(*~
	<docu>
		<summary>
			Completes the execution of the current step and moves the sequencer pointer to the next step in order of execution.
			The call returns ```ITcoObjectRestorer``` that allows to restore object upon step completition.
		</summary>		
		<returns></returns>	
	</docu>	
~*)
METHOD PROTECTED FINAL CompleteStep : ITcoObjectRestorer
_theOrderOfTheCurrentlyExecutedStep := _theOrderOfTheCurrentlyExecutedStep + 1;	
_currentStep.Status := eStepStatus.Done;
OnStepCompleted();
_modeController._stepIn.DoneWhen(_modeController._stepIn.Execute());
CompleteStep := THIS^;
END_METHOD

(*~
	<docu>
		<summary>
			Gets the information about the current step.						
		</summary>				
	</docu>	
~*)
PROPERTY CurrentStep : REFERENCE TO StepDetails
GET
CurrentStep REF= _currentStep;
END_GET
END_PROPERTY

METHOD FB_init : BOOL
VAR_INPUT
	bInitRetains : BOOL; // if TRUE, the retain variables are initialized (warm start / cold start)
	bInCopyCode : BOOL;  // if TRUE, the instance afterwards gets moved into the copy code (online change)
	Parent : ITcoObject;
	AutoRestoreMode : eRestoreMode; 
END_VAR
SUPER^.FB_init(bInitRetains, bInCopyCode, Parent, AutoRestoreMode);
END_METHOD

(*~
	<docu>
		<summary>
			Performs the check of the uniqueness of ```inStepId``` in the sequence.
			<remarks>			
				<note type="important">
					The StepId of each step in the sequence must be unique throughout the complete sequence, and it must not be changed.
				</note>
			</remarks>			
		</summary>				
	</docu>	
~*)
METHOD PRIVATE IsStepIdUnique
VAR_INPUT
(*~
	<docu>
		<summary>
			StepId to be checked for uniqueness.
		</summary>				
	</docu>	
~*)
	inStepID : INT;
END_VAR
VAR
	_i	: UINT;
	_hiIndex : UINT;
	_pUid : INT;
    _pNewSteps : POINTER TO INT;		
	_message : STRING(254);
END_VAR
IF ((_numberOfStepsInSequence <> _previousNumberOfStepsInSequence) AND _previousNumberOfStepsInSequence > 0) AND _stepIdUniquenessChecked AND NOT _sequencerHasError THEN
	_stepIdUniquenessChecked := FALSE;
	_previousNumberOfStepsInSequence := 0;
	_stepCounter := 0;
	_numberOfStepsInSequence := 0;
END_IF

IF NOT _stepIdUniquenessChecked AND NOT _sequencerHasError THEN

	// Increment order of the currently controlled step
	_theOrderOfTheCurrentlyEvaluatedStep := _theOrderOfTheCurrentlyEvaluatedStep + 1;
	
	IF(_stepCounter < _theOrderOfTheCurrentlyEvaluatedStep) THEN
		_stepCounter := _theOrderOfTheCurrentlyEvaluatedStep;
		_stepCounter := _stepCounter - 1; 
	END_IF
	
	_numberOfStepsInSequence := _stepCounter;
	
	IF (_numberOfStepsInSequence = _previousNumberOfStepsInSequence) AND (_numberOfStepsInSequence > 0) AND NOT _stepIdUniquenessChecked AND NOT _sequencerHasError THEN
		IF (_pPreviusSteps <> 0) THEN
			__DELETE(_pPreviusSteps);
		END_IF
		IF (_pNewSteps <> 0) THEN
			__DELETE(_pNewSteps);
		END_IF	
		_stepIdUniquenessChecked := TRUE;
		_theOrderOfTheCurrentlyEvaluatedStep := 0;
		_theOrderOfTheCurrentlyExecutedStep := 0;
		RETURN;		
	END_IF
	
	//Stores first StepId		
	IF (_numberOfStepsInSequence = 0) THEN
		//It should not exists, if yes delete and create again
		IF (_pPreviusSteps <> 0) THEN
			__DELETE(_pPreviusSteps);
		END_IF
		_pPreviusSteps := __NEW(UINT, 1);
		_pPreviusSteps[0] := inStepID;
	ELSE
		IF (_pNewSteps <> 0) THEN
			__DELETE(_pNewSteps);
		END_IF
		_pNewSteps := __NEW(UINT, (_numberOfStepsInSequence+1));

		//Compare with previous Steps and copy previous Steps to new array
		_hiIndex := _numberOfStepsInSequence-1;
		FOR _i := 0 TO _hiIndex DO
			_pUid := _pPreviusSteps[_i];
			IF inStepID = _pUid THEN
				IF NOT _sequencerHasError THEN
					IF (_pPreviusSteps <> 0) THEN
						__DELETE(_pPreviusSteps);
					END_IF	
					IF (_pNewSteps <> 0) THEN
						__DELETE(_pNewSteps);
					END_IF
					_sequencerErrorId := eSequencerError.NotUniqueStepId;
					_message := CONCAT('ERROR NOT UNIQUE STEP_ID ',UINT_TO_STRING(inStepID));
					_currentStep.Description := _message;
					_currentStep.Status := eStepStatus.Error;
					THIS^.Messenger.Post(_message, eMessageCategory.ProgrammingError);
					_sequencerHasError := TRUE;
					RETURN;					
				END_IF
			ELSE
				_pNewSteps[_i] := _pPreviusSteps[_i];
			END_IF
		END_FOR
		//Store new StepId
		_pNewSteps[_numberOfStepsInSequence] := inStepID;
		//Delete and create again
		IF (_pPreviusSteps <> 0) THEN
			__DELETE(_pPreviusSteps);
		END_IF		
		_pPreviusSteps :=  __NEW(UINT, (_numberOfStepsInSequence+1));
		//Copy
		_hiIndex := _hiIndex+1;
		FOR _i := 0 TO _hiIndex DO
			_pPreviusSteps[_i] := _pNewSteps[_i];			
		END_FOR

		IF (_pNewSteps <> 0) THEN
			__DELETE(_pNewSteps);
		END_IF
	END_IF	
END_IF
IF _stepIdUniquenessChecked THEN
	IF (_pPreviusSteps <> 0) THEN
		__DELETE(_pPreviusSteps);
	END_IF
	IF (_pNewSteps <> 0) THEN
		__DELETE(_pNewSteps);
	END_IF
END_IF
END_METHOD

(*~
	<docu>
		<summary>
			Main method of the sequener. Custom code needs to be placed here. The sequencer is executed by call of InstanceName.Run() method.
			This method is abstract, and it must be overridden in derived block.
		</summary>
	</docu>
~*)
METHOD PROTECTED ABSTRACT Main : BOOL
END_METHOD

(*~
	<docu>
		<summary>
			Handles changing the sequencer mode (Cyclic, Step).
		</summary>
	</docu>
~*)
PROPERTY ModeController : ITcoSequencerModeController
GET
ModeController := _modeController;
END_GET
END_PROPERTY

(*~
	<docu>
		<summary>
			Ensures that after each download, StepId uniqueness check is performed. 
			<remarks>			
				<note type="important">
					Do not call this method explicitly.
				</note>
			</remarks>		
		</summary>			
	</docu>	
~*)
{attribute 'call_after_online_change_slot' := '200'}
METHOD PRIVATE OnlineChange
_stepIdUniquenessChecked := FALSE;

_stepCounter := 0;
_numberOfStepsInSequence := 0;
_previousNumberOfStepsInSequence := 0;
END_METHOD


(*~
	<docu>
		<summary>
			This method is called on sequence completion (the sequencer's last step was completed). 
			This method can be overridden in derived block with a custom logic.
		</summary>			
	</docu>	
~*)
METHOD PROTECTED OnSequenceCompleted
END_METHOD

(*~
	<docu>
		<summary>
			This method is called when sequence enters error state. The method is called until the error is cleared. 
			This method can be overridden in derived block with a custom logic.
		</summary>			
	</docu>	
~*)
METHOD PROTECTED OnSequencerError
VAR_INPUT
	inErrorId : eSequencerError;
END_VAR
END_METHOD

(*~
	<docu>
		<summary>
			This method is executed upon step completion.
			This method can be overridden in derived block by custom logic.
		</summary>			
	</docu>	
~*)
METHOD PROTECTED OnStepCompleted
END_METHOD

(*~
	<docu>
		<summary>
			Implicit calling of this method is ensured by calling the method Run().
			It must not be called explicitely by consumer code in derived blocks.
			<remarks>			
				<note type="important">
					Do not call this method explicitly.
				</note>
			</remarks>
		</summary>			
	</docu>	
~*)
METHOD INTERNAL FINAL Open
VAR
	_message	:	STRING(254);
END_VAR
_theOrderOfTheCurrentlyEvaluatedStep := 0;

IF _requestStepActive AND _requestedStepId <> MinStepID AND (_modeController.Mode <> eSequencerMode.StepMode OR _modeController._stepIn.Busy OR _checkStepIdRequestedInStepMode) THEN
	_requestStepCycle := _requestStepCycle +1;
ELSE
	_requestStepCycle := 0;
END_IF

IF _requestStepCycle > 1 AND NOT _sequencerHasError THEN
	_sequencerErrorId := eSequencerError.StepWithRequestedIdDoesNotExists;
	_message := CONCAT('REQUESTED STEP_ID: ',UINT_TO_STRING(_requestedStepId));
	_message := CONCAT(_message, ' DOES NOT EXIST');
	_currentStep.Description := _message;
	_currentStep.Status := eStepStatus.Error;
	THIS^.Messenger.Post(_message, eMessageCategory.ProgrammingError);
	_sequencerHasError := TRUE;
END_IF

//???? Check if needs to be here.
IF _sequencerHasError AND (_sequencerErrorId = eSequencerError.NotUniqueStepId) THEN
	_sequencerErrorId := eSequencerError.noerror;	
	_sequencerHasError := FALSE;
	_stepIdUniquenessChecked := FALSE;
	_numberOfStepsInSequence := 0;
	_stepCounter := 0;
	_previousNumberOfStepsInSequence := 0;
END_IF

_restoringSequence := FALSE;
END_METHOD

(*~
	<docu>
		<summary>
			Terminates the currently executed step and set the sequencer's pointer to the step with Id that corresponds to ```inRequestedStepID``` parameter.
			When the order of the requested step is higher than the order of the currently finished step (the requested step is "after" the current one)
			the requested step is started in the same context cycle.
			When the order of the requested step is lower than the order of the currently finished step (the requested step is "before" the current one)
			the requested step is started in the next context cycle.
			If the requested step is not found even in the next context cycle, the sequencer enters error state ```StepWithRequestedIdDoesNotExists```.
			<para>
				See <see cref="eSequencerError"/> for detailed description.
			</para>
		</summary>
	</docu>
~*)
METHOD PROTECTED FINAL RequestStep : ITcoSequencer
VAR_INPUT
	(*~
		<docu>
			<summary>
				StepId of the step to be executed.
			</summary>
		</docu>
	~*)
	inRequestedStepID : INT := MinStepID;
END_VAR
VAR
	_message : STRING(254);
END_VAR
_modeController._stepIn.Restore();

_currentStep.Status := eStepStatus.Done;

_checkStepIdRequestedInStepMode := TRUE;

IF(inRequestedStepID <> MinStepID) THEN
	IF _requestedStepId <> MinStepID THEN
		IF NOT  _sequencerHasError THEN
			_sequencerErrorId := eSequencerError.MultipleRequestStepMethodCall;
			_message := CONCAT('REQUESTED STEP_ID: ',UINT_TO_STRING(inRequestedStepID));
			_message := CONCAT(_message, ' HAS BEEN REQUIRED, WHILE PREVIOUS REQUESTED STEP_ID: ');
			_message := CONCAT(_message,UINT_TO_STRING(_requestedStepId));
			_message := CONCAT(_message, ' HAS NOT BEEN YET PERFORMED!');
			_currentStep.Description := _message;
			_currentStep.Status := eStepStatus.Error;
			THIS^.Messenger.Post(_message, eMessageCategory.ProgrammingError);
			_sequencerHasError := TRUE;
		END_IF
	ELSE
		_requestStepCycle := 0;
		_requestedStepId := inRequestedStepID;
		_requestStepActive := TRUE;
	END_IF
END_IF;	

RequestStep := THIS^;
END_METHOD

(*~
	<docu>
		<summary>
			<para>
				This method resets the sequencer. 
				Method is typically called before starting the sequence or after error has occured in the sequence.
			</para>
		</summary>			
	</docu>	
~*)
METHOD PUBLIC Restore : ITcoRestorable
_restoringSequence := TRUE;

StepChanged(0);

_requestStepActive := FALSE;	
_requestedStepId := MinStepID;
_requestStepCycle := 0;
_sequencerHasError := FALSE;
_sequencerErrorId := eSequencerError.noError;
_currentStep.Description := '--------------------------';
_currentStep.ID := 0;
_currentStep.Order := 0;
_currentStep.Status := eStepStatus.None;
_currentStep.Duration := T#0S;

_stepCounter := 0;
_IdOfThePreviouslyExecutedStep := 0;
_numberOfStepsInSequence := 0;
_previousNumberOfStepsInSequence := 0;
_theOrderOfTheCurrentlyExecutedStep := 0;
_theOrderOfThePreviouslyExecutedStep := 0;
_stepIdUniquenessChecked := FALSE;

_StepIdChanged := FALSE;
_StepOrderChanged := FALSE;
_ChangeStepIdFrom := 0;
_ChangeStepIdTo := 0;
_ChangeStepOrderFrom := 0;
_ChangeStepOrderTo := 0;

_StepTimer(IN:= FALSE);

IF _modeController.Mode = eSequencerMode.Invalid THEN
	_modeController.Mode := eSequencerMode.CyclicMode;
END_IF

_modeController._stepForward.Restore();
_modeController._stepBackward.Restore();
_modeController._stepIn.Restore(); 	
_checkStepIdRequestedInStepMode := FALSE;
END_METHOD

(*~
	<docu>
		<summary>
			<para>
				Ensures calling the Open(), Main() and Close() methods in the desired order.
				This method is final, so it cannot be overloaded. The InstanceName.Run() needs to be called cyclically inside the appropriate context.
			</para>
		</summary>			
	</docu>	
~*)
METHOD PUBLIC FINAL Run
THIS^.Open();

_lastActiveCycle := Context.StartCycleCount; 

THIS^.Main();



IF _sequencerHasError THEN
	OnSequencerError(_sequencerErrorId);
END_IF
THIS^.Close();
END_METHOD

(*~
	<docu>
		<summary>
				Step of the sequence. 
		</summary>			
		<returns>
			True when step with given ```StepId``` is in order of the execution; the step is enabled and the sequencer is in the cyclic mode.
			True when step with given ```StepId``` is in order of the execution; the step is enabled, the sequencer is in the step mode and StepIn() method has been triggered.  			
		</returns>			
	</docu>	
~*)
METHOD PROTECTED FINAL Step : BOOL
VAR_INPUT
(*~
	<docu>
		<summary>
			StepId of the current step.
			<remarks>			
				<note type="important">
					This number must be unique throughout the complete sequence.
					It must be a constant or numerical literal and it must not change during the life-time of the sequencer. 
				</note>
			</remarks>
		</summary>		
	</docu>	
~*)
	inStepID				: 	INT;
(*~
	<docu>
		<summary>
			If this value is false, step body is not executed and execution is moved to the next enabled step.
		</summary>				
	</docu>	
~*)
	inEnabled				: 	BOOL;
(*~
	<docu>
		<summary>
			Step description text.
		</summary>				
	</docu>	
~*)
	inStepDescription		: 	STRING(254);		
END_VAR
VAR
	_message 				:	STRING(254);	
	_isInOrderOfExecution 	:	BOOL;	
	_stepModeActive 		: 	BOOL;
	_stepInExecuting 		: 	BOOL;
END_VAR
Step := FALSE;
IF inStepID <= MinStepID THEN
		_message := CONCAT('STEP_ID TOO LOW: ',INT_TO_STRING(inStepID));
		_message := CONCAT(_message, '! MINIMAL VALUE POSSIBLE: ');
		_message := CONCAT(_message,INT_TO_STRING(MinStepID + 1));
		_message := CONCAT(_message,'!!!');
		_currentStep.Description := _message;
		_currentStep.Status := eStepStatus.Error;
		THIS^.Messenger.Post(_message, eMessageCategory.ProgrammingError);
		_sequencerErrorId := eSequencerError.StepIdTooLow;
		_sequencerHasError := TRUE;
ELSIF  inStepID >= MaxStepID THEN
		_message := CONCAT('STEP_ID TOO HIGH: ',INT_TO_STRING(inStepID));
		_message := CONCAT(_message, '! MAXIMAL VALUE POSSIBLE: ');
		_message := CONCAT(_message,INT_TO_STRING(MaxStepID - 1));
		_message := CONCAT(_message,'!!!');
		_currentStep.Description := _message;
		_currentStep.Status := eStepStatus.Error;
		THIS^.Messenger.Post(_message, eMessageCategory.ProgrammingError);
		_sequencerErrorId := eSequencerError.StepIdTooHigh;
		_sequencerHasError := TRUE;
ELSIF NOT _sequencerHasError THEN
	Step := StepInternal(inStepID,inEnabled,inStepDescription);
END_IF;
END_METHOD

(*~
	<docu>
		<summary>
			This method is called at each transition between steps. 
		</summary>			
	</docu>	
~*)
METHOD PRIVATE StepChanged
VAR_INPUT
	newState : INT;
END_VAR
_isFirstStepEntry := TRUE;
_theOrderOfThePreviouslyExecutedStep := 0;
_IdOfThePreviouslyExecutedStep := MinStepID;

_StepTimer(IN:= FALSE);

SUPER^.ChangeStateProtected(newState);
END_METHOD

(*~
	<docu>
		<summary>
			Completes the actually running step, when the ```inCondition``` parameter is ```TRUE```.
			Method is typically called inside a step as the transition method.
		</summary>			
	</docu>	
~*)
METHOD PROTECTED FINAL StepCompleteWhen 
VAR_INPUT
(*~
	<docu>
		<summary>
			The condition under which the step is completed.
		</summary>			
	</docu>	
~*)
	inCondition : BOOL;
END_VAR
IF(inCondition) THEN
	THIS^.CompleteStep();
END_IF
END_METHOD

(*~
	<docu>
		<summary>
				Basic step of the sequence. 
		</summary>			
		<returns>
			True in case when step with given StepId is in order of the execution, the step is enabled and the sequencer is in the cyclic mode.
			True in case when step with given StepId is in order of the execution, the step is enabled, the sequencer is in the step mode and StepIn() method was triggered.  			
		</returns>			
	</docu>	
~*)
METHOD PRIVATE StepInternal : BOOL
VAR_INPUT
(*~
	<docu>
		<summary>
			StepId of the current step.
			<remarks>			
				<note type="important">
					This number must be unique throughout the complete sequence.
					It must be a constant or numerical literal and it must not change during the life-time of the sequencer. 
				</note>
			</remarks>
		</summary>		
	</docu>	
~*)
	inStepID				: 	INT;
(*~
	<docu>
		<summary>
			If this value is false, step body is not executed and execution is moved to the next enabled step.
		</summary>				
	</docu>	
~*)
	inEnabled				: 	BOOL;
(*~
	<docu>
		<summary>
			Step description text.
		</summary>				
	</docu>	
~*)
	inStepDescription		: 	STRING(254);		
END_VAR
VAR
	_message 				:	STRING(254);	
	_isInOrderOfExecution 	:	BOOL;	
	_stepModeActive 		: 	BOOL;
	_stepInExecuting 		: 	BOOL;
END_VAR
IF _modeController.Mode = eSequencerMode.Invalid THEN
	IF NOT _sequencerHasError THEN
		_currentStep.Description := 'INVALID MODE OF THE SEQUENCER!!!';
		_currentStep.Status := eStepStatus.Error;
		THIS^.Messenger.Post('INVALID MODE OF THE SEQUENCER!!!', eMessageCategory.Error);
		_sequencerErrorId := eSequencerError.InvalidSequencerMode;
		_sequencerHasError := TRUE;
	END_IF;		
	RETURN;
END_IF	

//-----------------------------------------------
//     		MULTIPLE CALL REGION
//-----------------------------------------------
// Initialize
StepInternal := FALSE;
_isFirstStepEntry := FALSE;
//-------------------------------------------------------------------------------------------------
//     		Check uniqueness of the StepId
//			If there are even two same StepIds or sequence has not been yet 
//			checked, method return FALSE, so no entrance to the step will be executed
//-------------------------------------------------------------------------------------------------
//-------------------------------------------------------------------------------------------------
//In case of call Restore() in OnStateChange(), this method must exits
//otherwise we get page fault
IF _restoringSequence THEN
	RETURN;
END_IF
IsStepIDUnique(inStepID);
IF NOT _stepIdUniquenessChecked THEN
	_theOrderOfThePreviouslyExecutedStep := -1;
	RETURN;
END_IF
//-------------------------------------------------------------------------------------------------
//-------------------------------------------------------------------------------------------------
// Cycle time measurement
_cycleTimer(IN:= TRUE, PT:= T#48D40H62M47S295MS);	
_SequenceElapsedTime  := _cycleTimer.ET;

// Specific step request
IF(_requestStepActive) AND (_requestedStepId = inStepID) AND (_theOrderOfTheCurrentlyEvaluatedStep >= 0) THEN
	_currentStep.Status := eStepStatus.Done;
	_theOrderOfTheCurrentlyExecutedStep 	:=	_theOrderOfTheCurrentlyEvaluatedStep;
	_theOrderOfThePreviouslyExecutedStep	:=	_theOrderOfTheCurrentlyExecutedStep;
	_requestedStepId := MinStepID;
	_requestStepCycle := 0;
	_requestStepActive := FALSE;
	StepChanged(_requestedStepId);
	//In case of call Restore() in OnStateChange(), this method must exits
	//otherwise we get page fault
	IF NOT _stepIdUniquenessChecked THEN
		StepInternal := FALSE;
		RETURN;
	END_IF								
END_IF
IF(_requestStepActive) THEN
	_theOrderOfTheCurrentlyEvaluatedStep := _theOrderOfTheCurrentlyEvaluatedStep + 1;
	RETURN;
END_IF

// STEP MODE COORDINATION
_stepModeActive := _modeController.Mode = eSequencerMode.StepMode;
_modeController(inCurrentStepRunning := _currentStep.Status = eStepStatus.Running);
IF(_stepModeActive) THEN			
	// StepForward
	IF _modeController._stepForward.Execute() THEN
		_modeController._stepIn.Restore();
		_modeController._stepBackward.Restore();
		IF _theOrderOfTheCurrentlyExecutedStep < _numberOfStepsInSequence THEN
			_theOrderOfTheCurrentlyExecutedStep := _theOrderOfTheCurrentlyExecutedStep + 1;
			_modeController._stepForward.DoneWhen(TRUE);
		ELSE
			_modeController._stepForward.Restore();
		END_IF			
	END_IF

	// Step Backward
	IF _modeController._stepBackward.Execute() THEN
		_modeController._stepIn.Restore();
		_modeController._stepForward.Restore();
		IF _theOrderOfTheCurrentlyExecutedStep > 0 THEN
			_theOrderOfTheCurrentlyExecutedStep := _theOrderOfTheCurrentlyExecutedStep - 1;
			_modeController._stepBackward.DoneWhen(TRUE);
		ELSE
			_modeController._stepForward.Restore();
		END_IF			
	END_IF			
END_IF;

IF(_modeController._stepForward.Done) THEN 
	_modeController._stepForward.Restore();
END_IF
IF(_modeController._stepBackward.Done) THEN
	_modeController._stepBackward.Restore();
END_IF		

// Determine the step is in order of execution
_isInOrderOfExecution := (_theOrderOfTheCurrentlyExecutedStep =_theOrderOfTheCurrentlyEvaluatedStep);

//-----------------------------------------------
//     		SINGLE PER STEP CALL REGION
//-----------------------------------------------
//Check if the order of the last executed step, has been changed  
IF(NOT _isInOrderOfExecution AND inStepID = _IdOfThePreviouslyExecutedStep) THEN
	IF _theOrderOfThePreviouslyExecutedStep <>_theOrderOfTheCurrentlyEvaluatedStep AND NOT _StepOrderChanged THEN
		_StepOrderChanged := TRUE;
		_ChangeStepOrderFrom := _theOrderOfThePreviouslyExecutedStep;
		_ChangeStepOrderTo := _theOrderOfTheCurrentlyEvaluatedStep;
	END_IF
END_IF

//Distinguish if StepId or step order has been changed 
IF (_theOrderOfTheCurrentlyEvaluatedStep >= _stepCounter) AND _StepIdChanged OR _StepOrderChanged THEN
	IF _StepOrderChanged AND NOT _StepIdChanged THEN
		_message := CONCAT('ERROR, STEP ORDER CHANGED DURING STEP EXECUTION FROM: ',UINT_TO_STRING(_ChangeStepOrderFrom));
		_message := CONCAT(_message , '=>');
		_message := CONCAT(_message , UINT_TO_STRING(_ChangeStepOrderTo));
		_currentStep.Description := _message;
		_currentStep.Status := eStepStatus.Error;
		THIS^.Messenger.Post(_currentStep.Description, eMessageCategory.ProgrammingError);
		_sequencerErrorId := eSequencerError.OrderOfTheStepHasBeenChanged;
	ELSIF _StepOrderChanged AND _StepIdChanged AND (_ChangeStepOrderFrom = _ChangeStepIdTo)  AND (_ChangeStepOrderTo = _ChangeStepIdFrom) THEN
		_message := CONCAT('ERROR, STEP ORDER CHANGED DURING STEP EXECUTION FROM: ',UINT_TO_STRING(_ChangeStepOrderFrom));
		_message := CONCAT(_message, '=>');
		_message := CONCAT(_message, UINT_TO_STRING(_ChangeStepOrderTo));
		_currentStep.Description := _message;
		_currentStep.Status := eStepStatus.Error;

		THIS^.Messenger.Post(_currentStep.Description, eMessageCategory.ProgrammingError);
		_sequencerErrorId := eSequencerError.OrderOfTheStepHasBeenChanged;
	ELSIF NOT _StepOrderChanged AND _StepIdChanged THEN
		_message := CONCAT('ERROR STEP_ID CHANGED DURING STEP EXECUTION FROM: ',UINT_TO_STRING(_ChangeStepIdFrom));
		_message := CONCAT(_message, '=>');
		_message := CONCAT(_message, UINT_TO_STRING(_ChangeStepIdTo));
		_currentStep.Description := _message;
		_currentStep.Status := eStepStatus.Error;

		THIS^.Messenger.Post(_currentStep.Description, eMessageCategory.ProgrammingError);
		_sequencerErrorId := eSequencerError.StepIdHasBeenChanged;
	ELSIF _StepOrderChanged AND _StepIdChanged AND (_ChangeStepOrderFrom = _ChangeStepIdFrom)  AND (_ChangeStepOrderTo = _ChangeStepIdTo) THEN
		_message := CONCAT('ERROR STEP_ID CHANGED DURING STEP EXECUTION FROM: ',UINT_TO_STRING(_ChangeStepIdFrom));
		_message := CONCAT(_message, '=>');
		_message := CONCAT(_message, UINT_TO_STRING(_ChangeStepIdTo));
		_currentStep.Description := _message;
		_currentStep.Status := eStepStatus.Error;

		THIS^.Messenger.Post(_currentStep.Description, eMessageCategory.ProgrammingError);
		_sequencerErrorId := eSequencerError.StepIdHasBeenChanged;
	END_IF
	_sequencerHasError := TRUE;
END_IF

IF NOT _isInOrderOfExecution AND _StepIdChanged THEN
	_theOrderOfTheCurrentlyEvaluatedStep := _theOrderOfTheCurrentlyEvaluatedStep + 1;
END_IF

IF (_StepOrderChanged OR _StepIdChanged OR _sequencerHasError) THEN
	RETURN;
END_IF

IF(_isInOrderOfExecution  AND NOT(_currentStep.Status = eStepStatus.Error)) THEN
	_currentStep.Status := eStepStatus.ReadyToRun;
	// Step is in the order of the execution, but it is disabled 
	IF NOT inEnabled THEN
		_currentStep.Status := eStepStatus.Disabled;
	END_IF
	_stepInExecuting := _modeController._stepIn.Busy;
	
	IF(NOT inEnabled AND NOT _stepInExecuting AND NOT _stepModeActive) THEN				
		_theOrderOfTheCurrentlyExecutedStep := _theOrderOfTheCurrentlyExecutedStep + 1;		
	END_IF					

	IF _stepModeActive THEN
		IF _modeController._stepIn.Execute() THEN
			_stepInExecuting := TRUE;			
			// Skips the step when not enabled
			IF(NOT inEnabled) THEN
				_theOrderOfTheCurrentlyExecutedStep := _theOrderOfTheCurrentlyExecutedStep + 1;
				_modeController._stepIn.Restore();
			END_IF
		END_IF	
		_currentStep.ID := inStepID;
		_currentStep.Enabled := inEnabled;
		IF NOT inEnabled THEN
			_currentStep.Description := CONCAT('(*',inStepDescription);		
			_currentStep.Description := CONCAT(_currentStep.Description,'*)');		
		ELSE
			_currentStep.Description := CONCAT('(>',inStepDescription);		
			_currentStep.Description := CONCAT(_currentStep.Description,'<)');		
		END_IF
	END_IF	

	StepInternal := (NOT _stepModeActive OR _stepInExecuting) AND inEnabled AND NOT(_currentStep.Status = eStepStatus.Error);

	IF(StepInternal) THEN
		//First entry to step production
		IF(_theOrderOfThePreviouslyExecutedStep <> _theOrderOfTheCurrentlyExecutedStep) THEN
			_isFirstStepEntry := TRUE;
			StepChanged(inStepID);
			//In case of call Restore() in OnStateChange(), this method must exits
			//otherwise we get page fault
			IF NOT _stepIdUniquenessChecked THEN
				StepInternal := FALSE;
				RETURN;
			END_IF								
		END_IF;	

		IF NOT CheckStepID(inStepID,_stepModeActive,_stepInExecuting) THEN
			StepInternal := FALSE;
			_theOrderOfTheCurrentlyEvaluatedStep := _theOrderOfTheCurrentlyEvaluatedStep + 1;
			_currentStep.Status := eStepStatus.Error;
			RETURN;
		END_IF
		_StepTimer(IN:= StepInternal, PT:= T#48D);		
		_StepElapsedTime := _StepTimer.ET;

		_currentStep.ID := inStepID;
		_currentStep.Enabled := inEnabled;
		_currentStep.Description := inStepDescription;
		_currentStep.Duration:= _StepElapsedTime;
		
		_IdOfThePreviouslyExecutedStep := inStepID;
		_theOrderOfThePreviouslyExecutedStep := _theOrderOfTheCurrentlyExecutedStep;
		
		_currentStep.Status := eStepStatus.Running; 
		_currentStep.Order := _theOrderOfTheCurrentlyExecutedStep;
	END_IF
END_IF
//-----------------------------------------------
//     		CONTINUOUS CALL REGION
//-----------------------------------------------
// Increment flow number
_theOrderOfTheCurrentlyEvaluatedStep := _theOrderOfTheCurrentlyEvaluatedStep + 1;

IF(_stepCounter < _theOrderOfTheCurrentlyEvaluatedStep) THEN
	_stepCounter := _theOrderOfTheCurrentlyEvaluatedStep;
	_stepCounter := _stepCounter - 1; 
END_IF

_numberOfStepsInSequence := _stepCounter;
END_METHOD

END_FUNCTION_BLOCK

// POUs/Prototypes/TcoState/TcoStateExtendible
FUNCTION_BLOCK ABSTRACT TcoStateExtendible EXTENDS TcoStateBase

METHOD PROTECTED FINAL ChangeState : ITcoState
VAR_INPUT
	NewState : INT;
END_VAR
ChangeState := SUPER^.ChangeStateProtected(NewState);
END_METHOD

END_FUNCTION_BLOCK

// POUs/Prototypes/TcoSequencer/TcoSequencerModeController
(*~
		<docu>
			<summary>
				Provides switching between sequencer modes so as handling stepping tasks in the step mode.
			</summary>
		</docu>
~*)
FUNCTION_BLOCK TcoSequencerModeController EXTENDS TcoObject IMPLEMENTS ITcoSequencerModeController
VAR_INPUT
	inCurrentStepRunning : BOOL;
END_VAR

VAR
(*~
	<docu>
		<summary>
			When '''TRUE''', disables changing between the modes of the sequencer.
		</summary>			
	</docu>	
~*)
	{attribute addProperty Name "<#Changing mode disabled#>"}
	{attribute clr [ReadOnly()]}
	_DisableModeChanging : BOOL;
(*~
	<docu>
		<summary>
			When '''TRUE''' skipping steps of the sequencer using methods '''StepBackward()''' and '''StepForward()''' is disabled.
		</summary>			
	</docu>	
~*)	
	{attribute addProperty Name "<#Skipping steps disabled#>"}
	{attribute clr [ReadOnly()]}
	_DisableStepSkipping : BOOL;
(*~
	<docu>
		<summary>
			Triggers StepBackward task, that decrements current step (variable: <c> TcoSequencer._theOrderOfTheCurrentlyExecutedStep</c> ), in case the sequencer is in step mode, and the current step is greather than zero.
		</summary>			
	</docu>	
~*)
	{attribute addProperty Name "<#Step backward#>"}
	_stepBackward : TcoTask(THIS^);	
(*~
	<docu>
		<summary>
			Triggers StepIn task, that changes the current step status from ReadyToRun to Running. 
			This causes starting the execution of the body of the current step.
		</summary>			
	</docu>	
~*)
	{attribute addProperty Name "<#Step in#>"}
	_stepIn : TcoTask(THIS^);	
(*~
	<docu>
		<summary>
			Triggers StepForward task, that increment current step (variable: <c>TcoSequencer._theOrderOfTheCurrentlyExecutedStep</c> ), 
			in case the sequencer is in step mode, and the current step is lower than number of steps in th sequence (variable: <c>TcoSequencer._numberOfStepsInSequence</c> ).
		</summary>			
	</docu>	
~*)
	{attribute addProperty Name "<#Step forward#>"}
	_stepForward : TcoTask(THIS^);
(*~
	<docu>
		<summary>
			Toggles between cyclic mode and step mode if not disabled.
			<para>
				See <see cref="TcoSequencerModeController.DisableModeChanging()"/> for detailed description.
			</para>		
		</summary>	
	</docu>	
~*)
	{attribute addProperty Name "<#Change mode#>"}
	_changeMode	: TcoTask(THIS^);
(*~
	<docu>
		<summary>
			Current mode of the sequencer.
		</summary>			
	</docu>	
~*)
	{attribute addProperty Name "<#Mode#>"}
	{attribute clr [ReadOnly()]}
	_mode : eSequencerMode;
	{attribute 'hide'}
	_previousMode : eSequencerMode := eSequencerMode.Invalid;
END_VAR

THIS^._changeMode.Enabled := NOT _DisableModeChanging;

IF _changeMode.Execute() THEN
	IF Mode = eSequencerMode.CyclicMode THEN
		Mode :=	 eSequencerMode.StepMode;
		_changeMode.Restore();
		RETURN;
	END_IF
	IF Mode = eSequencerMode.StepMode THEN
		Mode :=	 eSequencerMode.CyclicMode;
		_changeMode.Restore();
		RETURN;
	END_IF
END_IF

ChangeMode();

IF _changeMode.Done OR _changeMode.Error THEN
	_changeMode.Restore();
END_IF

METHOD PRIVATE ChangeMode
IF _previousMode <> _mode THEN
	//Restore all stepping task on mode change
	_stepForward.Restore();
	_stepBackward.Restore();
	_stepIn.Restore(); 	
	_changeMode.Restore(); 	
	//Mode change from cyclic to step, enabling stepping tasks according to settings.
	IF _previousMode = eSequencerMode.CyclicMode AND _mode = eSequencerMode.StepMode THEN
		_stepBackward.Enabled := NOT THIS^._DisableStepSkipping;
		_stepIn.Enabled := TRUE;
		_stepForward.Enabled := NOT THIS^._DisableStepSkipping;
		//If current step was running at the moment of switching from cyclic to step, stepIn task is invoked.			
		IF inCurrentStepRunning THEN
			_stepIn.Invoke(); 	
		END_IF
	END_IF
	//Disabling stepping tasks in case of Cyclic mode.
	IF _mode = eSequencerMode.CyclicMode THEN
		_stepBackward.Enabled := FALSE;
		_stepIn.Enabled := FALSE; 
		_stepForward.Enabled := FALSE;
	END_IF		
	_previousMode := _mode;
	OnModeChange(_previousMode,_mode);
END_IF
END_METHOD

(*~
	<docu>
		<summary>
			When ```TRUE```, disables mode change. 
		</summary>		
	</docu>	
~*)	
PROPERTY DisableModeChanging : BOOL
GET
DisableModeChanging := _DisableModeChanging;
END_GET
SET
_DisableModeChanging := DisableModeChanging;
END_SET
END_PROPERTY

(*~
	<docu>
		<summary>
			When ```TRUE``` disables step skipping (```StepBackward()``` and ```StepForward()```).
		</summary>		
	</docu>	
~*)	
PROPERTY DisableStepSkipping : BOOL
GET
DisableStepSkipping := _DisableStepSkipping;
END_GET
SET
_DisableStepSkipping := DisableStepSkipping;
END_SET
END_PROPERTY

(*~
	<docu>
		<summary>
			Gets or sets the mode of the sequencer. 
		</summary>		
	</docu>	
~*)	
PROPERTY Mode : eSequencerMode
GET
Mode := _mode;
END_GET
SET
IF NOT _DisableModeChanging THEN
	_mode := Mode;
END_IF
END_SET
END_PROPERTY

(*~
	<docu>
		<summary>
			Executes when mode of the sequencer changes. 
		</summary>		
	</docu>	
~*)	
METHOD PROTECTED OnModeChange
VAR_INPUT
	PreviousMode	: eSequencerMode;
	NewMode 		: eSequencerMode;
END_VAR
END_METHOD

(*~
	<docu>
		<summary>			
			Moves the sequencers pointer to the previous step.		
		</summary>			
	</docu>	
~*)
METHOD PUBLIC FINAL StepBackward
_stepBackward.Invoke();
END_METHOD

(*~
	<docu>
		<summary>
			Moves the sequencers pointer to the next step.
		</summary>			
	</docu>	
~*)
METHOD PUBLIC FINAL StepForward
_stepForward.Invoke();
END_METHOD

(*~
	<docu>
		<summary>
			Executes the step at the current sequencer's pointer.
		</summary>			
	</docu>	
~*)
METHOD PUBLIC FINAL StepIn
_stepIn.Invoke();
END_METHOD

END_FUNCTION_BLOCK

// POUs/TestFixtures/_internals_TcoContext
{attribute 'hide'}
{attribute clr [ExcludeFromApiDocumentation()]}
FUNCTION_BLOCK ABSTRACT _internals_TcoContext EXTENDS TcoContext
VAR
	_probeCurrentCycleCount  : ULINT;	
	_probeRunRequiredCycles : ULINT;
	_testId : ULINT;
END_VAR

{attribute 'TcRpcEnable'}
METHOD PROTECTED FINAL _Close
THIS^.Close();
END_METHOD

METHOD _GetSynchParams : RtcSynchParams
_GetSynchParams := RtcPrg._RtcSynchParams;
END_METHOD

{attribute 'TcRpcEnable'}
METHOD PROTECTED FINAL _Open
THIS^.Open();
END_METHOD

{attribute 'TcRpcEnable'}
METHOD PROTECTED FINAL _rtcUpdate
THIS^._rtc.Update();
END_METHOD

METHOD ProbeRun
IF(_probeCurrentCycleCount < _probeRunRequiredCycles) THEN 
	SUPER^.Run();	
	_probeCurrentCycleCount := _probeCurrentCycleCount + 1;
END_IF;
END_METHOD

END_FUNCTION_BLOCK

// POUs/TestFixtures/_internals_TcoSequencer
{attribute 'hide'}
{attribute clr [ExcludeFromApiDocumentation()]}
FUNCTION_BLOCK ABSTRACT _internals_TcoSequencer EXTENDS TcoSequencer

{attribute 'hide'}
METHOD PROTECTED FINAL _Close
THIS^.Close();
END_METHOD

{attribute 'hide'}
METHOD PROTECTED FINAL _Open
THIS^.Open();
END_METHOD

END_FUNCTION_BLOCK

// POUs/Utilities/StringBuilder
(*~
<docu>
	<summary>
			Allows to concat strings using fluent interface. It's similar to C# StringBuilder class
			Usage as follows :
			<code>
				ErrorString := _stringBuilder
					.Clear()
					.Append('Error number: ')
					.Append(INT_TO_STRING(ErrorNumber))
					.Append('. Message: ')
					.Append(ErrorMessage)
					.Append('.')
					.ToString();
			</code>
			
			Inspired by Gerhard Barteling blogpost at https://www.plccoder.com/fluent-code/
	</summary>				
</docu>	
~*)	
FUNCTION_BLOCK StringBuilder
VAR
	{attribute 'hide'}
    _workString:STRING;
END_VAR

METHOD Append : REFERENCE TO StringBuilder
VAR_INPUT
    Text :STRING; 
END_VAR
_workString := Concat(_workString,text);
Append REF= THIS^;
END_METHOD

METHOD Clear : REFERENCE TO StringBuilder
_workString := '';
Clear REF= THIS^;
END_METHOD

METHOD ToString : STRING
ToString := _workString;
END_METHOD

END_FUNCTION_BLOCK
